{attribute 'reflection'}
FUNCTION_BLOCK FB_Counter IMPLEMENTS I_Counter
VAR_INPUT
    bEnable : BOOL;
END_VAR
VAR_OUTPUT
    nCount : DINT;
END_VAR
VAR
    nStep : DINT := 1;
    nLimit : DINT := 100;
    nResets : INT;
END_VAR

IF bEnable THEN
    Increment();
END_IF

METHOD PUBLIC Increment : BOOL
VAR
    nNext : DINT;
END_VAR
nNext := nCount + nStep;
IF nNext > nLimit THEN
    nNext := nLimit;
END_IF
nCount := nNext;
Increment := nCount = nLimit;
END_METHOD

PROPERTY PUBLIC Step : DINT
GET
Step := nStep;
END_GET
SET
IF Step > 0 THEN
    nStep := Step;
END_IF
END_SET
END_PROPERTY

PROPERTY AtLimit : BOOL
GET
AtLimit := nCount >= nLimit;
END_GET
END_PROPERTY

ACTION Reset:
nCount := 0;
nResets := nResets + 1;
END_ACTION

END_FUNCTION_BLOCK

(* stored: Version 1.1.0.1, ProductVersion 3.1.4024.12
   POU FB_Counter: Id {5f1c2d9e-0a6b-4c11-9d3e-7a1b2c3d4e01}, SpecialFunc None
   Method Increment: Id {5f1c2d9e-0a6b-4c11-9d3e-7a1b2c3d4e02}
   Property Step: Id {5f1c2d9e-0a6b-4c11-9d3e-7a1b2c3d4e03}
   Get Get: Id {5f1c2d9e-0a6b-4c11-9d3e-7a1b2c3d4e04}
   Set Set: Id {5f1c2d9e-0a6b-4c11-9d3e-7a1b2c3d4e05}
   Property AtLimit: Id {5f1c2d9e-0a6b-4c11-9d3e-7a1b2c3d4e06}
   Get Get: Id {5f1c2d9e-0a6b-4c11-9d3e-7a1b2c3d4e07}
   Action Reset: Id {5f1c2d9e-0a6b-4c11-9d3e-7a1b2c3d4e08} *)
